{attribute 'GeneratedUsingTerminal: EJ7211-0010-0030'}
{attribute addProperty BoxType "EJ7211-0010-0030"}
{attribute addProperty Id "EtcSlaveTerminalBaseFB_PositionAT %I*FB_Position_3FA094ED4DRV_StatuswordAT %I*DRV_Statusword_9B36FDFC2DRV_ControlwordAT %Q*DRV_Controlword_F3F147212DRV_Target_velocityAT %Q*DRV_Target_velocity_08A9583B4WcStateAT %I*WcState_9091E0EB2InfoDataAT %I*InfoData_6185D47C20"}
{attribute addProperty CRC "3497715898"}
{attribute addProperty Size "34"}
TYPE EJ7211_D07AE8BA EXTENDS EtcSlaveTerminalBase :
STRUCT
	{attribute addProperty Name "FB_Position"}
	FB_Position : FB_Position_3FA094ED;
	{attribute addProperty Name "DRV_Statusword"}
	DRV_Statusword : DRV_Statusword_9B36FDFC;
	{attribute addProperty Name "DRV_Controlword"}
	DRV_Controlword : DRV_Controlword_F3F14721;
	{attribute addProperty Name "DRV_Target_velocity"}
	DRV_Target_velocity : DRV_Target_velocity_08A9583B;
	{attribute addProperty Name "WcState"}
	WcState : WcState_9091E0EB;
	{attribute addProperty Name "InfoData"}
	InfoData : InfoData_6185D47C;
END_STRUCT
END_TYPE

(* stored: Version 1.2.0.0, ProductVersion 3.1.4024.9
   DUT EJ7211_D07AE8BA: Id {8f1918ba-2732-45e3-aee8-d7af0f2a156d} *)
